(* CODESYS project 3.2GearInDyn.project

Project tree, tasks and I/O mapping:
  Device : CODESYS SoftMotion Win V3 x64, 3S - Smart Software Solutions GmbH, version 3.5.12.0
    application Application
      libraries: Standard, * (System); VisuDialogs, * (System)
      task MainTask (cyclic, interval t#2ms, priority 1) calls PLC_PRG
      task VISU_TASK (cyclic, interval 100 ms, priority 31) calls VisuElems.Visu_Prg
      program PLC_PRG [ST]
      visualisation Visualization
      trace Trace (task MainTask): AxisMaster.fActVelocity, AxisSlave.fActVelocity, AxisMaster.fActPosition, AxisSlave.fActPosition, AxisMaster.fActAcceleration, AxisSlave.fActAcceleration, PLC_PRG.mcGearInPos.Execute, PLC_PRG.mcGearInPos.InSync, PLC_PRG.mcGearInPos.Busy, PLC_PRG.mcGearInPos.StartSync, AxisMaster.fSetPosition, AxisSlave.fSetPosition
      function block MC_GearInDyn [ST]
      visualisation MC_GearInDyn
      visualisation Visualization_1
    SoftMotion General Axis Pool
      AxisMaster : SM_Drive_Virtual, 3S - Smart Software Solutions GmbH, order no. 1805, version 4.0.0.0
          settings: wDriveID = 0; iMovementType = 0
      AxisSlave : SM_Drive_Virtual, 3S - Smart Software Solutions GmbH, order no. 1805, version 4.0.0.0
          settings: iMovementType = 0
  text list GlobalTextList
  text list AxisStatus
*)

// Device/Application/PLC_PRG
PROGRAM PLC_PRG
VAR
	//定义Master主轴相关的功能块
	mcPMaster  		:  MC_Power ;
	mcMoveVelocity  : MC_MoveVelocity ;
	mcStopMaster  	: MC_stop;
	mcResetM         : MC_Reset;
	//定义从轴相关功能块；
	mcPSlave    : MC_Power ;
	mcStopSlave : MC_Stop ;
	mcResetS      : MC_Reset;
	mcSetPostion  : MC_SetPosition;
	//Gear 
	mcGearIn  	: MC_GearIn ;
	mcGearOut  	: MC_GearOut ;
	mcGearInPos : MC_GearInPos;
	
	mcGearInDyn  : MC_GearInDyn ;
	//辅助变量
	bGearIn   	: BOOL;
	bStartMove  : BOOL;
END_VAR

//主轴和从轴的使能
mcPMaster(
	Axis:= AxisMaster, 
	Enable:= TRUE , 
	bRegulatorOn:= TRUE , 
	bDriveStart:=TRUE , 
	Status=> , 
	bRegulatorRealState=> , 
	bDriveStartRealState=> , 
	Busy=> , 
	Error=> , 
	ErrorID=> );
mcPSlave(
	Axis:= AxisSlave , 
	Enable:= TRUE, 
	bRegulatorOn:= TRUE , 
	bDriveStart:= TRUE, 
	Status=> , 
	bRegulatorRealState=> , 
	bDriveStartRealState=> , 
	Busy=> , 
	Error=> , 
	ErrorID=> );
//齿轮耦合
mcGearIn(
	Master:= AxisMaster, 
	Slave:= AxisSlave, 
	Execute:= , 
	RatioNumerator:= , 
	RatioDenominator:= , 
	Acceleration:= , 
	Deceleration:= , 
	Jerk:= , 
	InGear=> , 
	Busy=> , 
	CommandAborted=> , 
	Error=> , 
	ErrorID=> );
//动态耦合
mcGearInDyn(
	Execute:= , 
	fRatio:= , 
	Acceleration:= , 
	Deceleration:= , 
	Jerk:= , 
	InGear=> , 
	Busy=> , 
	CommandAborted=> , 
	Error=> , 
	ErrorID=> , 
	Master:= AxisMaster, 
	Slave:= AxisSlave  );
mcGearInPos(
	Master:= AxisMaster, 
	Slave:= AxisSlave, 
	Execute:= , 
	RatioNumerator:= , 
	RatioDenominator:= , 
	MasterSyncPosition:= , 
	SlaveSyncPosition:= , 
	MasterStartDistance:= , 
	AvoidReversal:= , 
	StartSync=> , 
	InSync=> , 
	Busy=> , 
	CommandAborted=> , 
	Error=> , 
	ErrorID=> );
mcGearOut(
	Slave:=AxisSlave , 
	Execute:= , 
	Done=> , 
	Busy=> , 
	Error=> , 
	ErrorID=> );	
//主轴开始运动
mcMoveVelocity(
	Axis:=AxisMaster , 
	Execute:=  , 
	Velocity:= , 
	Acceleration:= 100, 
	Deceleration:= 100, 
	Jerk:= , 
	Direction:= , 
	InVelocity=> , 
	Busy=> , 
	CommandAborted=> , 
	Error=> , 
	ErrorID=> );
	
//停止
mcStopMaster(
	Axis:= AxisMaster, 
	Execute:= , 
	Deceleration:= , 
	Jerk:= , 
	Done=> , 
	Busy=> , 
	Error=> , 
	ErrorID=> );
mcStopSlave(
	Axis:= AxisSlave, 
	Execute:= , 
	Deceleration:= , 
	Jerk:= , 
	Done=> , 
	Busy=> , 
	Error=> , 
	ErrorID=> );
mcSetPostion(
	Axis:= AxisSlave, 
	Execute:= , 
	Position:= , 
	Mode:= , 
	Done=> , 
	Busy=> , 
	Error=> , 
	ErrorID=> );	
//复位
mcResetM(
	Axis:= AxisMaster, 
	Execute:= , 
	Done=> , 
	Busy=> , 
	Error=> , 
	ErrorID=> );
mcResetS(
	Axis:= AxisSlave, 
	Execute:= , 
	Done=> , 
	Busy=> , 
	Error=> , 
	ErrorID=> );

END_PROGRAM

// Device/Application/MC_GearInDyn
FUNCTION_BLOCK MC_GearInDyn
VAR_INPUT
	Execute : BOOL;//触发,上升沿有效
	fRatio  : LREAL := 1.0;//比例系数,负数代表反向耦合
	Acceleration : LREAL;
	Deceleration : LREAL;
	Jerk         : LREAL;
END_VAR
VAR_OUTPUT
	InGear  : BOOL;
	Busy    : BOOL;
	CommandAborted : BOOL;
	Error   : BOOL;
	ErrorID : SMC_Error;
END_VAR
VAR
	mcGearIN  : MC_GearIn;
	rtrigExe  : R_TRIG;
	fLastRatio  : LREAL;
END_VAR
VAR_IN_OUT
	Master : AXIS_REF_SM3;
	Slave  : AXIS_REF_SM3;
END_VAR

rtrigExe(clk:=Execute);
IF rtrigExe.Q THEN
	IF fRatio <> fLastRatio AND fRatio <> 0 THEN
		fLastRatio := fRatio;
		mcGearIN.RatioNumerator :=TO_DINT( fRatio * 10000);
		mcGearIn.RatioDenominator := 10000;
		mcGearIN.Execute := TRUE;
	END_IF
END_IF
IF Slave.nAxisState <> smc_aXIS_sTATE.synchronized_motion THEN
	fLastRatio := 0;
END_IF
mcGearIN(
	Master:= Master, 
	Slave:= Slave, 
	Execute:= , 
	RatioNumerator:= , 
	RatioDenominator:= , 
	Acceleration:= Acceleration, 
	Deceleration:= Deceleration, 
	Jerk:= Jerk, 
	InGear=> InGear, 
	Busy=> Busy, 
	CommandAborted=> CommandAborted, 
	Error=> Error, 
	ErrorID=> ErrorID);
	
mcGearIN.Execute := FALSE;

END_FUNCTION_BLOCK

// Device/Application/Visualization
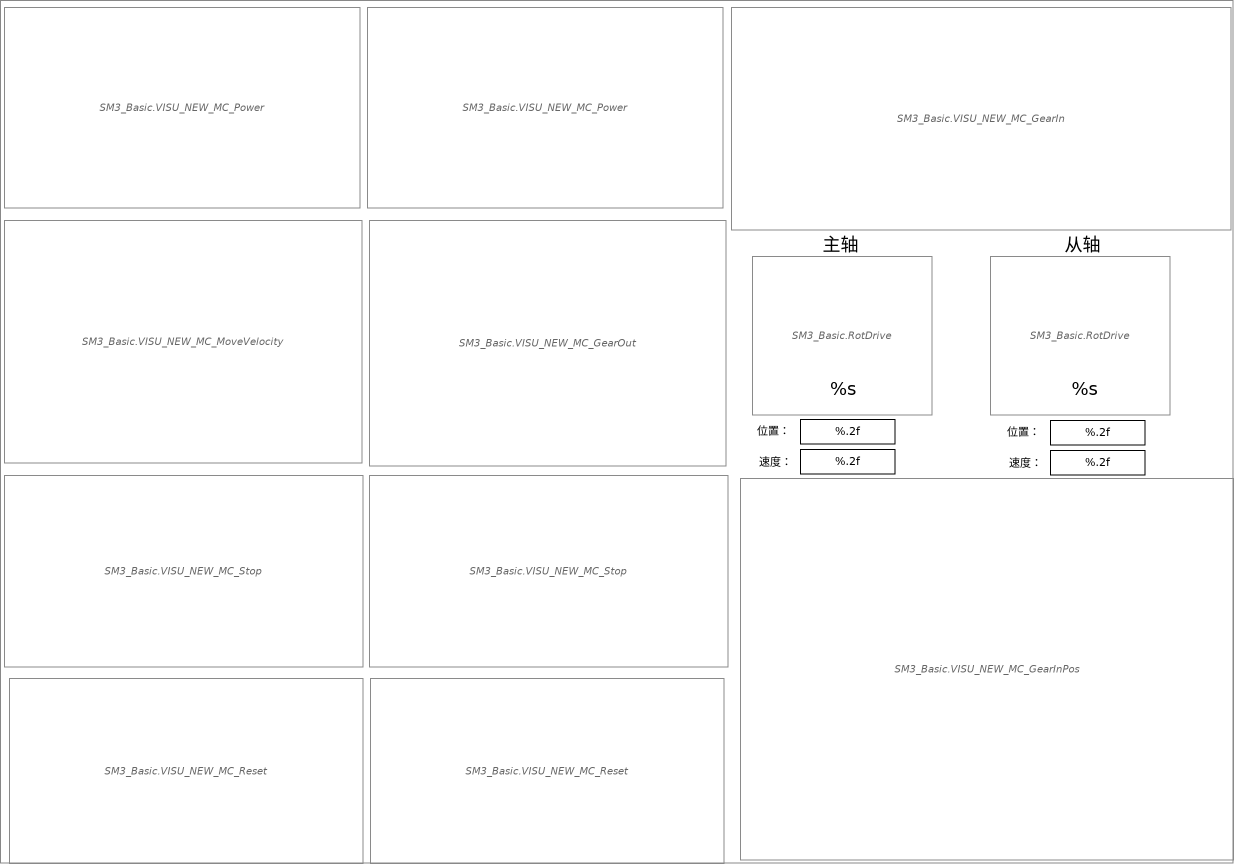
VISUALIZATION Visualization  // 1234x864
    Frame (4,7 356x201)
        shows SM3_Basic.VISU_NEW_MC_Power(m_Input_FB := PLC_PRG.mcPMaster)
    Frame (367,7 356x201)
        shows SM3_Basic.VISU_NEW_MC_Power(m_Input_FB := PLC_PRG.mcPSlave)
    Frame (4,220 358x243)
        shows SM3_Basic.VISU_NEW_MC_MoveVelocity(m_Input_FB := PLC_PRG.mcMoveVelocity)
    Frame (4,475 359x192)
        shows SM3_Basic.VISU_NEW_MC_Stop(m_Input_FB := PLC_PRG.mcStopMaster)
    Frame (369,475 359x192)
        shows SM3_Basic.VISU_NEW_MC_Stop(m_Input_FB := PLC_PRG.mcStopSlave)
    Frame (369,220 357x246)
        shows SM3_Basic.VISU_NEW_MC_GearOut(m_Input_FB := PLC_PRG.mcGearOut)
    Frame (731,7 500x223)
        shows SM3_Basic.VISU_NEW_MC_GearIn(m_Input_FB := PLC_PRG.mcGearIn)
    Frame (752,256 180x159)
        shows SM3_Basic.RotDrive(m_Input_AXISREF := Axismaster)
    Frame (990,256 180x159)
        shows SM3_Basic.RotDrive(m_Input_AXISREF := AxisSlave)
    Frame (9,678 354x186)
        shows SM3_Basic.VISU_NEW_MC_Reset(m_Input_FB := PLC_PRG.mcResetM)
    Frame (370,678 354x186)
        shows SM3_Basic.VISU_NEW_MC_Reset(m_Input_FB := PLC_PRG.mcResetS)
    Frame (740,478 494x382)
        shows SM3_Basic.VISU_NEW_MC_GearInPos(m_Input_FB := PLC_PRG.mcGearInPos)
    Label (793,230 95x30), "主轴"
    Label (1035,230 95x30), "从轴"
    Label (734,416 79x30), "位置："
    Label (736,447 79x30), "速度："
    Rectangle (800,419 95x25), "%.2f", text variable: AxisMaster.fActPosition
    Rectangle (800,449 95x25), "%.2f", text variable: AxisMaster.fActVelocity
    Label (986,448 79x30), "速度："
    Label (984,417 79x30), "位置："
    Rectangle (1050,420 95x25), "%.2f", text variable: AxisSlave.fActPosition
    Rectangle (1050,450 95x25), "%.2f", text variable: AxisSlave.fActVelocity
    Rectangle (738,374 211x30), "%s", text list: 'AxisStatus', text index: AxisMaster.nAxisState
    Rectangle (978,374 214x30), "%s", text list: 'AxisStatus', text index: AxisSlave.nAxisState
END_VISUALIZATION

// Device/Application/MC_GearInDyn
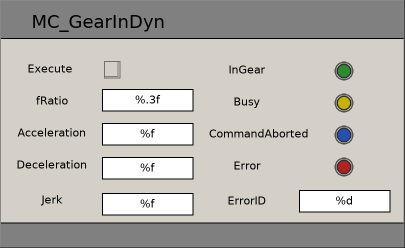
VISUALIZATION MC_GearInDyn  // 405x248
VAR_IN_OUT
	m_Input_FB : MC_GearInDyn ;
END_VAR
    RoundedRectangle (0,0 405x248)
    Rectangle (0,38 405x185)
    Label (8,7 181x30), "MC_GearInDyn"
    Label (7,54 90x30), "Execute"
    Label (7,86 90x30), "fRatio"
    Label (7,150 90x30), "Deceleration"
    Label (7,118 90x30), "Acceleration"
    Label (7,185 90x30), "Jerk"
    Button (104,61 16x17)
        toggle m_Input_FB.Execute
    Rectangle (102,89 91x22), "%.3f", text variable: m_Input_FB.fRatio
        OnMouseClick: write the text variable via Default
    Rectangle (102,123 91x22), "%f", text variable: m_Input_FB.Acceleration
        OnMouseClick: write the text variable via Default
    Rectangle (102,157 91x22), "%f", text variable: m_Input_FB.Deceleration
        OnMouseClick: write the text variable via Default
    Rectangle (102,193 91x22), "%f", text variable: m_Input_FB.Jerk
        OnMouseClick: write the text variable via Default
    Label (202,87 90x30), "Busy"
    Label (202,55 90x30), "InGear"
    Label (202,151 90x30), "Error"
    Label (202,119 114x30), "CommandAborted"
    Label (202,186 90x30), "ErrorID"
    Lamp1 (333,60 22x22), variable: m_Input_FB.InGear, style: Lamp-Lamp1-Green
    Lamp1 (333,92 22x22), variable: m_Input_FB.Busy, style: Lamp-Lamp1-Yellow
    Lamp1 (333,124 22x22), variable: m_Input_FB.CommandAborted, style: Lamp-Lamp1-Blue
    Lamp1 (333,156 22x22), variable: m_Input_FB.Error, style: Lamp-Lamp1-Red
    Rectangle (299,190 91x22), "%d", text variable: m_Input_FB.ErrorID
END_VISUALIZATION

// Device/Application/Visualization_1
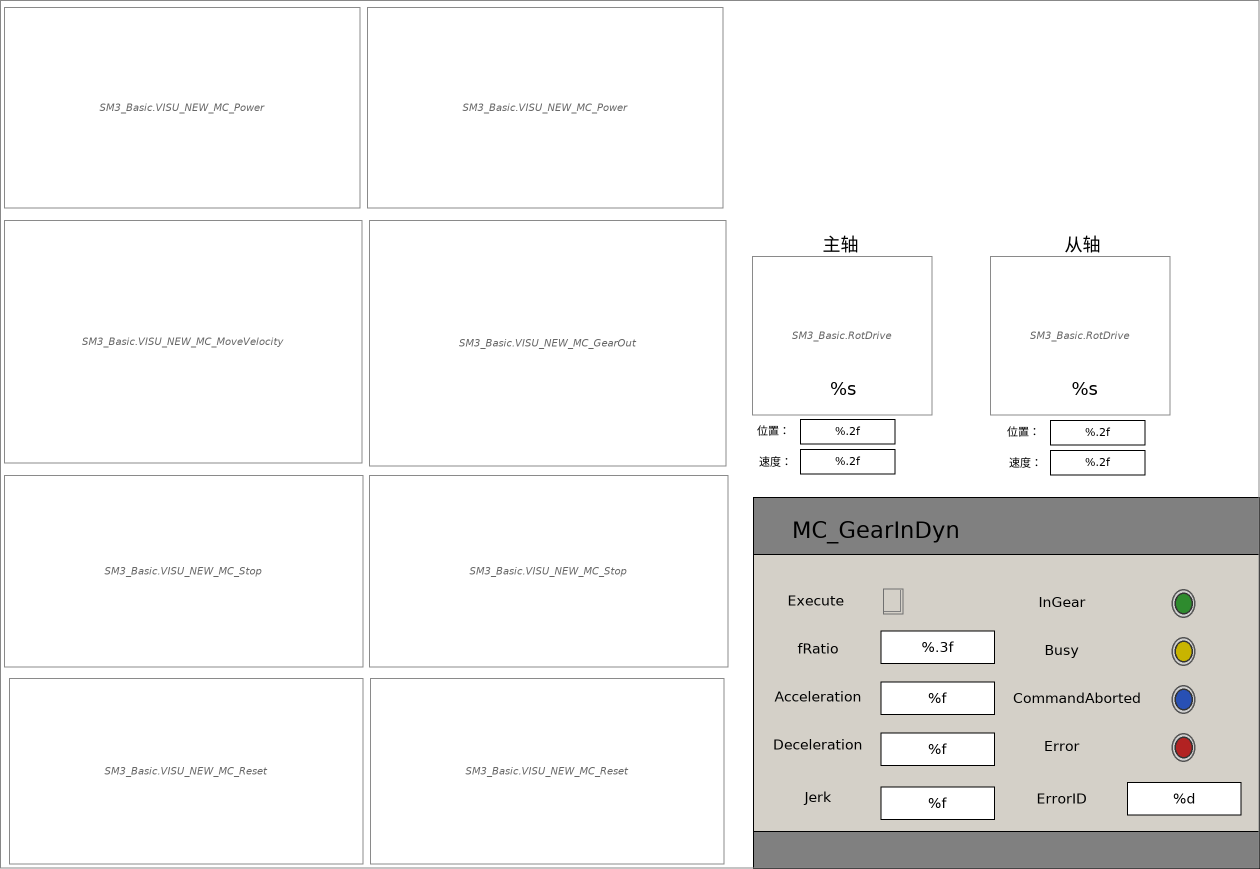
VISUALIZATION Visualization_1  // 1260x869
    Frame (4,7 356x201)
        shows SM3_Basic.VISU_NEW_MC_Power(m_Input_FB := PLC_PRG.mcPMaster)
    Frame (367,7 356x201)
        shows SM3_Basic.VISU_NEW_MC_Power(m_Input_FB := PLC_PRG.mcPSlave)
    Frame (4,220 358x243)
        shows SM3_Basic.VISU_NEW_MC_MoveVelocity(m_Input_FB := PLC_PRG.mcMoveVelocity)
    Frame (4,475 359x192)
        shows SM3_Basic.VISU_NEW_MC_Stop(m_Input_FB := PLC_PRG.mcStopMaster)
    Frame (369,475 359x192)
        shows SM3_Basic.VISU_NEW_MC_Stop(m_Input_FB := PLC_PRG.mcStopSlave)
    Frame (369,220 357x246)
        shows SM3_Basic.VISU_NEW_MC_GearOut(m_Input_FB := PLC_PRG.mcGearOut)
    Frame (752,256 180x159)
        shows SM3_Basic.RotDrive(m_Input_AXISREF := Axismaster)
    Frame (990,256 180x159)
        shows SM3_Basic.RotDrive(m_Input_AXISREF := AxisSlave)
    Frame (9,678 354x186)
        shows SM3_Basic.VISU_NEW_MC_Reset(m_Input_FB := PLC_PRG.mcResetM)
    Frame (370,678 354x186)
        shows SM3_Basic.VISU_NEW_MC_Reset(m_Input_FB := PLC_PRG.mcResetS)
    Label (793,230 95x30), "主轴"
    Label (1035,230 95x30), "从轴"
    Label (734,416 79x30), "位置："
    Label (736,447 79x30), "速度："
    Rectangle (800,419 95x25), "%.2f", text variable: AxisMaster.fActPosition
    Rectangle (800,449 95x25), "%.2f", text variable: AxisMaster.fActVelocity
    Label (986,448 79x30), "速度："
    Label (984,417 79x30), "位置："
    Rectangle (1050,420 95x25), "%.2f", text variable: AxisSlave.fActPosition
    Rectangle (1050,450 95x25), "%.2f", text variable: AxisSlave.fActVelocity
    Rectangle (738,374 211x30), "%s", text list: 'AxisStatus', text index: AxisMaster.nAxisState
    Rectangle (978,374 214x30), "%s", text list: 'AxisStatus', text index: AxisSlave.nAxisState
    Frame (753,497 507x372)
        shows MC_GearInDyn(m_Input_FB := PLC_PRG.mcGearInDyn)
END_VISUALIZATION

(* text list AxisStatus (id | default)
  0 | power_off
  1 | errorstop
  2 | stopping
  3 | standstill
  4 | discrete_motion
  5 | continuous_motion
  6 | synchronized_motion
  7 | homing
   |  *)
